DATA_BLOCK "MB_CLIENT_DB"
{InstructionName := 'MB_CLIENT';
 LibVersion := '5.1';
 S7_Optimized_Access := 'TRUE' }
AUTHOR : SIMATIC
FAMILY : MBUS_TCP
NAME : MB_CLI
VERSION : 5.1
NON_RETAIN
MB_CLIENT

BEGIN

END_DATA_BLOCK

